// TwinCAT 3 PLC project PLC1
// ProgramVersion: 3.1.4024.0
// libraries:
//   SPT Vision, * (Beckhoff Automation LLC)
//   Tc2_Standard, * (Beckhoff Automation GmbH)
//   Tc2_System, * (Beckhoff Automation GmbH)
//   Tc3_Module, * (Beckhoff Automation GmbH)
//   Tc3_Vision, * (Beckhoff Automation GmbH)
// project tree:
//   / GlobalTextList.TcGTLO (not stored), PlcTask.TcTTO (not stored), Visualization Manager.TcVMO (not stored)
//   POUs/ FB_ImageAquire.TcPOU (not stored), MAIN.TcPOU
//   VISUs/ V_Main.TcVIS

// ---- POUs/MAIN.TcPOU
PROGRAM MAIN
VAR
	Camera1 : FB_ImageAquire; 


	Playback : FB_ImageToVideo := (CameraName 			:= 'Camera1', 
							   	   JsonAttribute 		:= '{CreateVid : 1, CameraName: "Camera1"}', 
							   	   FramesPerSecond 		:= 10,
							   	   TimeBeforeEvent		:= T#7S,
								   TimeAfterEvent		:= T#3S,
								   VideoOutputDirectory := 'C:\TcAlarmVideo',
								   ReductionFactor 		:= 0.25);

	TriggerEvent : BOOL;
END_VAR

Camera1.CyclicLogic();
IF Camera1.ImageAvailable THEN
	Playback.AddImage(ipImageIn := Camera1.Image);
END_IF

Playback.CyclicLogic();
IF TriggerEvent THEN
	TriggerEvent := FALSE;
	Playback.TriggerAlarmForVideoCapture();
END_IF

END_PROGRAM

// ---- VISUs/V_Main.TcVIS
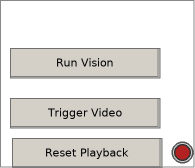
VISUALIZATION V_Main  // 195x168
    Button (10,48 150x30), "Run Vision"
        toggle MAIN.Camera1.RunVision
    Button (10,98 150x30), "Trigger Video"
        toggle MAIN.TriggerEvent
    Button (12,138 150x30), "Reset Playback"
        tap MAIN.Playback._Reset
    Lamp1 (170,140 25x25), variable: MAIN.Playback._Error, style: Lamp-Lamp1-Red
END_VISUALIZATION
